{attribute 'GeneratedUsingTerminal: EK1121-0010-0016'}
{attribute addProperty BoxType "EK1121-0010-0016"}
{attribute addProperty Id "EtcSlaveTerminalBaseInfoDataAT %I*InfoData_6F19DB2B2"}
{attribute addProperty CRC "2874840167"}
{attribute addProperty Size "2"}
TYPE EK1121_AB5A9467 EXTENDS EtcSlaveTerminalBase :
STRUCT
	{attribute addProperty Name "InfoData"}
	InfoData : InfoData_6F19DB2B;
END_STRUCT
END_TYPE

(* stored: Version 1.2.0.0, ProductVersion 3.1.4024.9
   DUT EK1121_AB5A9467: Id {f3cd5d68-48a3-4f62-bd91-664255a4bdee} *)
